MOVL C09996 V=800.0 PL=0
CALL JOB:DEMO_ROOF_SIDE_0625_3PAINT_60
END
